{attribute 'GeneratedUsingTerminal: EL2521-0000-1019'}
{attribute addProperty BoxType "EL2521-0000-1019"}
{attribute addProperty Id "PTO_StatusAT %I*PTO_Status_40B3051C7ENC_Status_compactAT %I*ENC_Status_compact_036460C97PTO_ControlAT %Q*PTO_Control_9287F8E45PTO_Target_compactAT %Q*PTO_Target_compact_5C359F7D2ENC_Control_compactAT %Q*ENC_Control_compact_2ED727EF3WcStateAT %I*WcState_9091E0EB2InfoDataAT %I*InfoData_94A18F5E2"}
{attribute addProperty CRC "890439464"}
{attribute addProperty Size "28"}
TYPE EL2521_35130728 EXTENDS EtcSlaveTerminalBase_947E5A46 :
STRUCT
	{attribute addProperty Name "PTO_Status"}
	PTO_Status : PTO_Status_40B3051C;
	{attribute addProperty Name "ENC_Status_compact"}
	ENC_Status_compact : ENC_Status_compact_036460C9;
	{attribute addProperty Name "PTO_Control"}
	PTO_Control : PTO_Control_9287F8E4;
	{attribute addProperty Name "PTO_Target_compact"}
	PTO_Target_compact : PTO_Target_compact_5C359F7D;
	{attribute addProperty Name "ENC_Control_compact"}
	ENC_Control_compact : ENC_Control_compact_2ED727EF;
	{attribute addProperty Name "WcState"}
	WcState : WcState_9091E0EB;
	{attribute addProperty Name "InfoData"}
	InfoData : InfoData_94A18F5E;
END_STRUCT
END_TYPE

(* stored: Version 1.2.0.0, ProductVersion 3.1.4024.9
   DUT EL2521_35130728: Id {b2c2be5f-06f3-4d65-ad53-a8d2123750f8} *)
